{attribute 'GeneratedUsingTerminal: ELX1054-0000-0016'}
{attribute addProperty BoxType "ELX1054-0000-0016"}
{attribute addProperty Description "ELX1054 4Ch. Dig. Input NAMUR, NO/NC, Ex i"}
{attribute addProperty Physics "KK"}
{attribute addProperty Id "Channel_1AT %I*Channel_31CEFA7F2Channel_2AT %I*Channel_31CEFA7F2Channel_3AT %I*Channel_31CEFA7F2Channel_4AT %I*Channel_31CEFA7F2Input_Type_NCAT %I*Input_Type_NC_5EE695414WcStateAT %I*WcState_9091E0EB2InfoDataAT %I*InfoData_6F19DB2B2"}
{attribute addProperty CRC "4014447438"}
{attribute addProperty Size "16"}
TYPE ELX1054_EF479B4E EXTENDS EtcSlaveTerminalBase_947E5A46 :
STRUCT
	{attribute addProperty Name "Channel_1"}
	Channel_1 : Channel_31CEFA7F;
	{attribute addProperty Name "Channel_2"}
	Channel_2 : Channel_31CEFA7F;
	{attribute addProperty Name "Channel_3"}
	Channel_3 : Channel_31CEFA7F;
	{attribute addProperty Name "Channel_4"}
	Channel_4 : Channel_31CEFA7F;
	{attribute addProperty Name "Input_Type_NC"}
	Input_Type_NC : Input_Type_NC_5EE69541;
	{attribute addProperty Name "WcState"}
	WcState : WcState_9091E0EB;
	{attribute addProperty Name "InfoData"}
	InfoData : InfoData_6F19DB2B;
END_STRUCT
END_TYPE

(* stored: Version 1.2.0.0, ProductVersion 3.1.4024.11
   DUT ELX1054_EF479B4E: Id {be84c124-597e-4315-86a7-3ddc08fbc9da} *)
